TYPE ST_Record :
STRUCT
    bEnabled   : BOOL;
    nValue     : INT;
    rScale     : REAL;
    sLabel     : STRING;
END_STRUCT
END_TYPE

(* stored: Version 1.1.0.1, ProductVersion 3.1.4024.10 *)
